Universal Robots PolyScope program: End-to-end_Accuracy_Check.urp

Program TagAccuracy (installation=calibgrid directory=/programs/Tutorials createdIn=5.11.6 lastSavedIn=5.17.1 robotSerialNumber=20205500252)
Calibrated DH parameters: a=[0.000184, -0.219652, -0.392286, 0.000038, 0.000028, 0]; d=[0.162619, 336.622473, -336.554151, 0.064764, 0.099721, 0.099645]; alpha=[1.568905, 0.001082, 0.006941, 1.569865, -1.571178, 0]; deltaTheta=[0, 1.028123, 5.256271, -0.001213, 0, 0]
InitVariablesNode
Robot Program (runOnlyOnce=false)
  MoveJ speed 60 deg/s, acceleration 80 deg/s^2 (useActiveTCP=true) feature=Base
    Waypoint Waypoint_1: TCP in base x=234.215 y=196.378 z=163.39 mm, rx=2.8369 ry=-1.3082 rz=-0.0078 rad; joints [65.559, -83.461, -151.49, -36.029, 90.578, 25.311] deg
  URCap Roboception (rc_urcap, Roboception GmbH) dataModel(SENSOR=rc_visard 1, MODULE=AprilTag, FUNCTION=Detect)
  URCap Roboception (rc_urcap, Roboception GmbH) dataModel(SENSOR=rc_visard 1, MODULE=AprilTag, FUNCTION=GetPose, grasp_approach=Orientation from pick module, use_popup=true, Variable(key=STORE_POSE_VARIABLE, variable(name=pose_1)))
  URCap Roboception (rc_urcap, Roboception GmbH) dataModel(SENSOR=rc_visard 1, MODULE=AprilTag, FUNCTION=GetPose, grasp_approach=Orientation from pick module, use_popup=true, Variable(key=STORE_POSE_VARIABLE, variable(name=pose_2)))
  center := interpolate_pose(pose_1, pose_2, 0.5)
  above := pose_trans(center, p[0,0,-0.1,0,0,0])
  Popup Message (haltProgram=false message=center inputType=Variable) variable=center
  MoveL speed 250 mm/s, acceleration 1200 mm/s^2 (useActiveTCP=true) feature=Base
    Waypoint Variable (Variable): variable=above
    Waypoint Variable (Variable): motionParameters(jointSpeed=1.047198 jointAcceleration=1.396263 cartesianSpeed=0.05 cartesianAcceleration=1.2); variable=center
      Until TOOL_CONTACT_DETECTION (allowActions=false retraction=0.002 decelerationAcceleration=3 decelerationAngularAcceleration=34.906585)
    Popup Message (haltProgram=false message=continue? inputType=Text)
    Waypoint Variable (Variable): variable=above
